(*
Searches an `I_Entity` for a `I_StateManager` component matching provided id pattern.
Result:
- Ok - Returns `I_StateManager`.
- None - Returns null.
- Err.Itf0 - Returns null, incorrect interface.
*)
FUNCTION GetStateManager : Result
VAR_INPUT
	iEntity		: I_Entity;
END_VAR
VAR_OUTPUT
	iSmgr		: I_StateManager;
END_VAR
VAR
	i			: Iter(1);
	_iComp		: I_FatComponent;
	cmp			: TagCmp;
END_VAR

IF iEntity = 0 THEN
	GetStateManager := Err.Itf0;
	RETURN;
END_IF

WHILE IsOk(iEntity.Get(i.Next(), iComp => _iComp)) DO
	IF IsOk(ICompToIStateMgr(_iComp.Raw, iDest => iSmgr)) THEN
		GetStateManager := Ok;
		RETURN;
	END_IF
END_WHILE

END_FUNCTION

(* stored: Version 1.1.0.1
   POU GetStateManager: Id {cc9710d2-5f6d-4b85-a1d3-6aee9f41ddac}, SpecialFunc None *)
